// TwinCAT 3 PLC project Main
// ProgramVersion: 3.1.4024.0
// libraries:
//   Tc2_Standard, * (Beckhoff Automation GmbH)
//   Tc2_System, * (Beckhoff Automation GmbH)
//   Tc2_Utilities, * (Beckhoff Automation GmbH)
//   Tc3_Module, * (Beckhoff Automation GmbH)
//   TcUnit, * (www.tcunit.org)
//   [mobject-commands], * (mobject)
// project tree:
//   Programs/ DummyCommand.TcPOU, Main.TcPOU
//   Tasks/ PlcTask.TcTTO
// real-time tasks:
//   TASK PlcTask: cycle T#10ms, priority 20, ADS port 350

CONFIGURATION Main
    RESOURCE PLC ON TwinCAT3
        TASK PlcTask(INTERVAL := T#10ms, PRIORITY := 20);
        PROGRAM Main WITH PlcTask : Main;
    END_RESOURCE
END_CONFIGURATION

// ---- Programs/Main.TcPOU
PROGRAM Main
VAR
	// Standalone command execution
	pStandaloneCommand : POINTER TO DummyCommand;
	runStandaloneCommand : BOOL;
	abortStandaloneCommand : BOOL;
	simulateErrorStandaloneCommand : BOOL;
	simulatedStandaloneCommandErrorId : UDINT := 1234;
	
	standaloneCommandResult : I_Result;
	standaloneCommandCompleted : BOOL;
	standaloneCommandAborted : BOOL;
	standaloneCommandError : BOOL;
	standaloneCommandErrorId : UDINT;
	
	// SingleAsyncCommandRunner command execution
	
	// QueuedPoolAsyncCommandRunner command execution
	runQueuedPoolCommand : BOOL;
	pQueuedCommand : POINTER TO DummyCommand;

	queuedPoolCommandRunner : QueuedPoolAsyncCommandRunner(poolCapacity := 2, queueCapacity := 5);
	
	// Support variables
	id : DINT;
END_VAR

// Standalone command execution
IF runStandaloneCommand THEN
	runStandaloneCommand := FALSE;
	pStandaloneCommand := __NEW(DummyCommand(id := NextId(), name := 'standalone'));
END_IF

IF pStandaloneCommand <> 0 THEN
	IF pStandaloneCommand^.Idle THEN
		pStandaloneCommand^.Execute();
	ELSIF pStandaloneCommand^.Executing THEN
		pStandaloneCommand^.CyclicCall();
		
		IF abortStandaloneCommand THEN
			abortStandaloneCommand := FALSE;
			pStandaloneCommand^.Abort();
		END_IF
		
		IF simulateErrorStandaloneCommand THEN
			simulateErrorStandaloneCommand := FALSE;
			pStandaloneCommand^.SimulateError(simulatedStandaloneCommandErrorId);
		END_IF
	ELSIF pStandaloneCommand^.Stopped THEN
		standaloneCommandResult := pStandaloneCommand^.GetResult();
		__DELETE(pStandaloneCommand);
		standaloneCommandCompleted := standaloneCommandResult.Completed;
		standaloneCommandAborted := standaloneCommandResult.Aborted;
		standaloneCommandError := standaloneCommandResult.Error;
		standaloneCommandErrorId := standaloneCommandResult.ErrorId;
		standaloneCommandResult.Dispose();
		standaloneCommandResult := 0;
	END_IF
END_IF

// SingleAsyncCommandRunner command execution

// QueuedPoolAsyncCommandRunner command execution
IF runQueuedPoolCommand THEN
	runQueuedPoolCommand := FALSE;
	pQueuedCommand := __NEW(DummyCommand(id := NextId(), name := 'queued-pool'));
	queuedPoolCommandRunner.QueueCommand(pQueuedCommand^);
END_IF

queuedPoolCommandRunner.CyclicCall();

METHOD PRIVATE NextId : DINT
NextId := id;
id := id + 1;
END_METHOD

END_PROGRAM

// ---- Programs/DummyCommand.TcPOU
{attribute 'linkalways'} 
{attribute 'no_explicit_call' := 'This FB is a CLASS and must be accessed using methods or properties'}
{attribute 'enable_dynamic_creation'}
FUNCTION_BLOCK PUBLIC DummyCommand EXTENDS AsyncCommand
VAR
	id : DINT;
	name : T_MaxString;
	timer : Ton;
END_VAR

METHOD PRIVATE AdsLog
VAR_INPUT
	message : T_MaxString;
END_VAR
VAR
	arrghhhh : T_MaxString := '%s';
END_VAR
VAR_INST
	format : FB_FormatString;
END_VAR
format(
	sFormat := 'DummyCommand{id=%d, name=%s} -> %s',
	arg1 := F_DInt(id),
	arg2 := F_String(name),
	arg3 := F_String(arrghhhh)
);

AdsLogStr(
	msgCtrlMask := ADSLOG_MSGTYPE_HINT,
	msgFmtStr := format.sOut,
	strArg := message
);
END_METHOD

METHOD FB_init : BOOL
VAR_INPUT
	bInitRetains : BOOL; // if TRUE, the retain variables are initialized (warm start / cold start)
	bInCopyCode : BOOL;  // if TRUE, the instance afterwards gets moved into the copy code (online change)
	id : DINT;
	name : T_MaxString;
END_VAR
THIS^.id := id;
THIS^.name := name;

AdsLog('FB_init');
END_METHOD

METHOD PROTECTED OnAborted
AdsLog('Aborted');
END_METHOD

METHOD PROTECTED OnAborting
VAR_INPUT
	stateControl : I_AsyncCommandStateControl;
END_VAR
AdsLog('Aborting');

WrapItUp(stateControl);
END_METHOD

METHOD PROTECTED OnCompleted : BOOL
AdsLog('Completed');
END_METHOD

METHOD PROTECTED OnCompleting
VAR_INPUT
	stateControl : I_AsyncCommandStateControl;
END_VAR
AdsLog('Completing');

WrapItUp(stateControl);
END_METHOD

METHOD PROTECTED OnErrored
VAR_INST
	firstCycle : BOOL;
END_VAR
IF NOT firstCycle THEN
	firstCycle := TRUE;
	AdsLog('Errored');
END_IF
END_METHOD

METHOD PROTECTED OnExecuting
VAR_INPUT
	stateControl : I_AsyncCommandStateControl;
END_VAR
VAR_INST
	firstCycle : BOOL;
END_VAR
IF NOT firstCycle THEN
	firstCycle := TRUE;
	AdsLog('Executing');
END_IF

timer(IN := TRUE, PT := T#10S);
IF timer.Q THEN
	stateControl.Next();
END_IF
END_METHOD

METHOD PROTECTED OnIdle
VAR_INST
	firstCycle : BOOL;
END_VAR
IF NOT firstCycle THEN
	firstCycle := TRUE;
	AdsLog('Idle');
END_IF
END_METHOD

METHOD PROTECTED OnInitializing
VAR_INPUT
	stateControl : I_AsyncCommandStateControl;
END_VAR
AdsLog('Initialising');

stateControl.Next();
END_METHOD

METHOD PUBLIC SimulateError
VAR_INPUT
	errorId : UDINT;
END_VAR
stateMachine.Error(errorId);
END_METHOD

METHOD PRIVATE WrapItUp
VAR_INPUT
	stateControl : I_AsyncCommandStateControl;
END_VAR
timer(IN := FALSE);
stateControl.Next();
END_METHOD

END_FUNCTION_BLOCK
